// TIA Portal V19 export
TYPE "Prod_Pers"
   STRUCT
      Data : Struct
         MODE : "Prod_Mode";
         SET_UP : "Prod_SetUp_Data";
         INTERRUZIONI : "Prod_Interruzioni";
         Aspo_In_Linea_Prev_Values : "Coil_Item";
         Aspo_In_Carico_Prev_Values : "Coil_Item";
         Taglio_Finale_Prev_Values : "Coil_Item";
         "C_ID_Aspo_In_Linea_@AbortCut" { S7_SetPoint := 'True'} : DInt;
         "C_ID_Aspo_In_Linea_@CoilEnd" : DInt;
      END_STRUCT;
      Par : Struct
         MES_Operating : Int := 1;   // Funzionameto MES (0 = OFF; 1= ON)
         AUT_PushOrder_InProduction : Int := 1;   // Mette automaticamente gli ordini in produzione quando il precedente è concluso (0 = NO; 1 = SI)
         PartTolFactor_BAD_EXCEED_TOL : Real := 3.0;   // Fattore moltiplicativo su tolleranza lunghezza parte tagliata per assegnazione diretta NG e non TO_CHECK
         Material_To_Go_Additional : Real := 10000.0;
         Material_To_Go_Low_Speed : Real := 2000.0;
      END_STRUCT;
   END_STRUCT;
END_TYPE
